% RSLogix 500 project AT_Lab 1.RSS, saved by version 12.00.00.00 %
PROJECT "UNTITLED"    % processor: Bul.1763 MicroLogix 1100 Series A %

PROGRAM FILES
  LAD 2   4 rungs

DATA FILES
  O0 OUTPUT  4 elements
  I1 INPUT  6 elements
  S2 STATUS  66 elements
  B3 BINARY  1 elements
  T4 TIMER  2 elements
  C5 COUNTER  1 elements
  R6 CONTROL  1 elements
  N7 INTEGER  1 elements
  F8 FLOAT  1 elements

LADDER 2
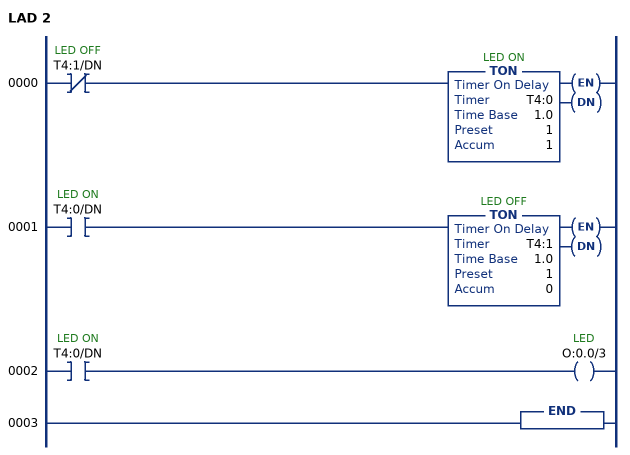
% Rung: 0 %
SOR XIO T4:1/DN TON T4:0 1.0 1 1 EOR
%   T4:1/DN  "LED OFF" %
%   T4:0  "LED ON" %
% Rung: 1 %
SOR XIC T4:0/DN TON T4:1 1.0 1 0 EOR
%   T4:0/DN  "LED ON" %
%   T4:1  "LED OFF" %
% Rung: 2 %
SOR XIC T4:0/DN OTE O:0.0/3 EOR
%   T4:0/DN  "LED ON" %
%   O:0.0/3  "LED" %
% Rung: 3 %
SOR END EOR

OTHER DOCUMENTED ADDRESSES
  O:0.0/0  "LED"
  O:0.0/1  "LED"

DATA TABLE (non-zero values as saved)
DATA T4
% .PRE .ACC %
% T4:0 % 1 1
% T4:1 % 1 0
